(* Logix 5000 project; controller EuniceF_ICA6 vendor 1 type 14 code 150 rev 37.11; software revision 37.00 *)

TASK MainTask (continuous, watchdog 500 ms) : MainProgram

MODULES
   Local : vendor 1 type 14 code 150 (Compact 0, rev 37.11)
      Discrete_IO : Embedded (Compact 1, rev 3.1, Output RPI 20 ms)
      Analog_IO : Embedded (Compact 2, rev 1.1, Output RPI 80 ms)
      Counters : Embedded (Compact 3, rev 1.1, Output RPI 20 ms)
END_MODULES

VAR_GLOBAL   (* controller tags *)
   COIL1 : ALIAS FOR Local:1:O.Data.3;
   COIL2 : ALIAS FOR Local:1:O.Data.2;
   HIGH : ALIAS FOR Local:1:I.Data.15;
   LOCK : ALIAS FOR Local:1:O.Data.1;
   RESET : ALIAS FOR Local:1:I.Data.12;
   START : ALIAS FOR Local:1:I.Data.11;
   STOP : ALIAS FOR Local:1:I.Data.13;
   VIB : ALIAS FOR Local:1:I.Data.14;
END_VAR

PROGRAM MainProgram   (* main routine MainRoutine *)

ROUTINE MainRoutine   (* ladder *)
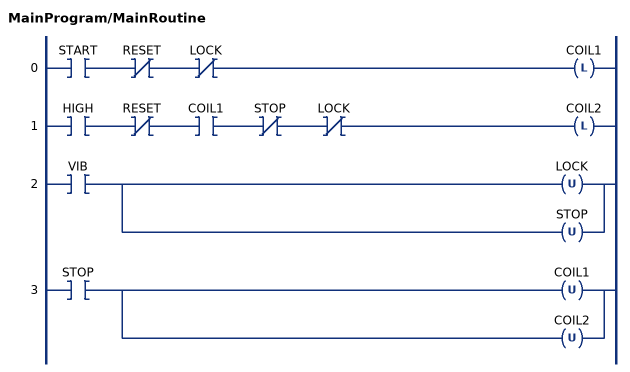
   0: XIC(START)XIO(RESET)XIO(LOCK)OTL(COIL1);
   1: XIC(HIGH)XIO(RESET)XIC(COIL1)XIO(STOP)XIO(LOCK)OTL(COIL2);
   2: XIC(VIB)[OTU(LOCK) ,OTU(STOP) ];
   3: XIC(STOP)[OTU(COIL1) ,OTU(COIL2) ];
END_ROUTINE
END_PROGRAM
